# B&R Automation Studio project NewPendant_NG4_11_05_25A (part 9)

```c
			break;

			case 1: // Pulse

				curCfg->Param[parTIG_AmpSP].segmYes = 1;
				curCfg->Param[parTIG_AmpInSP].segmYes = 0;
				curCfg->Param[parTIG_AmpOutSP].segmYes = 0;
				curCfg->Param[parTIG_BackAmp].segmYes = 1;
				curCfg->Param[parTIG_PulseFreq].segmYes = 1;
				curCfg->Param[parTIG_PulseWidth].segmYes = 1;

				switch(curCfg->Param_ENUM[parENUM_AVC_Mode].val[0]){

					default:

					curCfg->Param[parAVC_VoltSP].segmYes = 1;
					curCfg->Param[parAVC_VoltInSP].segmYes = 0;
					curCfg->Param[parAVC_VoltOutSP].segmYes = 0;
					curCfg->Param[parAVC_VoltBackSP].segmYes = 1;

					break;

					case 1: // BackGround Locked

					curCfg->Param[parAVC_VoltSP].segmYes = 1;
					curCfg->Param[parAVC_VoltInSP].segmYes = 0;
					curCfg->Param[parAVC_VoltOutSP].segmYes = 0;
					curCfg->Param[parAVC_VoltBackSP].segmYes = 0;

					break;

					case 2: // ForeGround Locked

					curCfg->Param[parAVC_VoltSP].segmYes = 0;
					curCfg->Param[parAVC_VoltInSP].segmYes = 0;
					curCfg->Param[parAVC_VoltOutSP].segmYes = 0;
					curCfg->Param[parAVC_VoltBackSP].segmYes = 1;

					break;

					case 3: // Locked

					curCfg->Param[parAVC_VoltSP].segmYes = 0;
					curCfg->Param[parAVC_VoltInSP].segmYes = 0;
					curCfg->Param[parAVC_VoltOutSP].segmYes = 0;
					curCfg->Param[parAVC_VoltBackSP].segmYes = 0;

					break;

				}

			break;

			case 2: // Synch

				curCfg->Param[parTIG_AmpSP].segmYes = 1;
				curCfg->Param[parTIG_AmpInSP].segmYes = 0;
				curCfg->Param[parTIG_AmpOutSP].segmYes = 0;
				curCfg->Param[parTIG_BackAmp].segmYes = 1;
				curCfg->Param[parTIG_PulseFreq].segmYes = 0;
				curCfg->Param[parTIG_PulseWidth].segmYes = 0;

				switch(curCfg->Param_ENUM[parENUM_AVC_Mode].val[0]){

					default:

					curCfg->Param[parAVC_VoltSP].segmYes = 1;
					curCfg->Param[parAVC_VoltInSP].segmYes = 0;
					curCfg->Param[parAVC_VoltOutSP].segmYes = 0;
					curCfg->Param[parAVC_VoltBackSP].segmYes = 1;

					break;

					case 1: // BackGround Locked

					curCfg->Param[parAVC_VoltSP].segmYes = 1;
					curCfg->Param[parAVC_VoltInSP].segmYes = 0;
					curCfg->Param[parAVC_VoltOutSP].segmYes = 0;
					curCfg->Param[parAVC_VoltBackSP].segmYes = 0;

					break;

					case 2: // ForeGround Locked

					curCfg->Param[parAVC_VoltSP].segmYes = 0;
					curCfg->Param[parAVC_VoltInSP].segmYes = 0;
					curCfg->Param[parAVC_VoltOutSP].segmYes = 0;
					curCfg->Param[parAVC_VoltBackSP].segmYes = 1;

					break;

					case 3: // Locked

					curCfg->Param[parAVC_VoltSP].segmYes = 0;
					curCfg->Param[parAVC_VoltInSP].segmYes = 0;
					curCfg->Param[parAVC_VoltOutSP].segmYes = 0;
					curCfg->Param[parAVC_VoltBackSP].segmYes = 0;

					break;

				}

			break;

			case 3: // Synch In/Out

				curCfg->Param[parTIG_AmpSP].segmYes = 0;
				curCfg->Param[parTIG_AmpInSP].segmYes = 1;
				curCfg->Param[parTIG_AmpOutSP].segmYes = 1;
				curCfg->Param[parTIG_BackAmp].segmYes = 1;
				curCfg->Param[parTIG_PulseFreq].segmYes = 0;
				curCfg->Param[parTIG_PulseWidth].segmYes = 0;

				switch(curCfg->Param_ENUM[parENUM_AVC_Mode].val[0]){

					default:

					curCfg->Param[parAVC_VoltSP].segmYes = 0;
					curCfg->Param[parAVC_VoltInSP].segmYes = 1;
					curCfg->Param[parAVC_VoltOutSP].segmYes = 1;
					curCfg->Param[parAVC_VoltBackSP].segmYes = 1;

					break;

					case 1: // BackGround Locked

					curCfg->Param[parAVC_VoltSP].segmYes = 0;
					curCfg->Param[parAVC_VoltInSP].segmYes = 1;
					curCfg->Param[parAVC_VoltOutSP].segmYes = 1;
					curCfg->Param[parAVC_VoltBackSP].segmYes = 0;

					break;

					case 2: // ForeGround Locked

					curCfg->Param[parAVC_VoltSP].segmYes = 0;
					curCfg->Param[parAVC_VoltInSP].segmYes = 0;
					curCfg->Param[parAVC_VoltOutSP].segmYes = 0;
					curCfg->Param[parAVC_VoltBackSP].segmYes = 1;

					break;

					case 3: // Locked

					curCfg->Param[parAVC_VoltSP].segmYes = 0;
					curCfg->Param[parAVC_VoltInSP].segmYes = 0;
					curCfg->Param[parAVC_VoltOutSP].segmYes = 0;
					curCfg->Param[parAVC_VoltBackSP].segmYes = 0;

					break;

					}

			break;

		}

		switch(_TVL_MODE){

			default: // Straight

				curCfg->Param[parTVL_VelSP].segmYes = 1;
				curCfg->Param[parTVL_VelInSP].segmYes = 0;
				curCfg->Param[parTVL_VelOutSP].segmYes = 0;
				curCfg->Param[parTVL_VelBackSP].segmYes = 0;

			break;

			case 1:

				curCfg->Param[parTVL_VelSP].segmYes = 1;
				curCfg->Param[parTVL_VelInSP].segmYes = 0;
				curCfg->Param[parTVL_VelOutSP].segmYes = 0;
				curCfg->Param[parTVL_VelBackSP].segmYes = 1;

			break;

			case 2:

				curCfg->Param[parTVL_VelSP].segmYes = 0;
				curCfg->Param[parTVL_VelInSP].segmYes = 1;
				curCfg->Param[parTVL_VelOutSP].segmYes = 1;
				curCfg->Param[parTVL_VelBackSP].segmYes = 1;

			break;

		}

		switch(_WF_MODE){

			default: // Straight

				curCfg->Param[parWF_SpeedSP].segmYes = 1;
				curCfg->Param[parWF_SpeedInSP].segmYes = 0;
				curCfg->Param[parWF_SpeedOutSP].segmYes = 0;
				curCfg->Param[parWF_BkgSpeedSP].segmYes = 0;

			break;

			case 1:

				curCfg->Param[parWF_SpeedSP].segmYes = 1;
				curCfg->Param[parWF_SpeedInSP].segmYes = 0;
				curCfg->Param[parWF_SpeedOutSP].segmYes = 0;
				curCfg->Param[parWF_BkgSpeedSP].segmYes = 1;

			break;

			break;

			case 2:

				curCfg->Param[parWF_SpeedSP].segmYes = 0;
				curCfg->Param[parWF_SpeedInSP].segmYes = 1;
				curCfg->Param[parWF_SpeedOutSP].segmYes = 1;
				curCfg->Param[parWF_BkgSpeedSP].segmYes = 1;

			break;

			break;

		}

		switch(_WP_MODE){

			default: // Straight

				curCfg->Param[parWP_SpeedSP].segmYes = 1;
				curCfg->Param[parWP_SpeedInSP].segmYes = 0;
				curCfg->Param[parWP_SpeedOutSP].segmYes = 0;
				curCfg->Param[parWP_BkgSpeedSP].segmYes = 0;

			break;

			case 1:

				curCfg->Param[parWP_SpeedSP].segmYes = 1;
				curCfg->Param[parWP_SpeedInSP].segmYes = 0;
				curCfg->Param[parWP_SpeedOutSP].segmYes = 0;
				curCfg->Param[parWP_BkgSpeedSP].segmYes = 1;

			break;

			break;

			case 2:

				curCfg->Param[parWP_SpeedSP].segmYes = 0;
				curCfg->Param[parWP_SpeedInSP].segmYes = 1;
				curCfg->Param[parWP_SpeedOutSP].segmYes = 1;
				curCfg->Param[parWP_BkgSpeedSP].segmYes = 1;

			break;

			break;

		}

		hmi->PLC_Changes |= 0xF;
		KK_Was_Cahnged = 1;
	}

	_TIG_Mode = curCfg->Param_ENUM[parENUM_TIG_Mode].val[0];

	_AVC_Mode = curCfg->Param_ENUM[parENUM_AVC_Mode].val[0];

	_TVL_SYN_MODE = curCfg->Param_ENUM[parENUM_TVL_SYN_MODE].val[0];

	_WF_SYN_MODE = curCfg->Param_ENUM[parENUM_WF_SYN_MODE].val[0];

	_WP_SYN_MODE = curCfg->Param_ENUM[parENUM_WP_SYN_MODE].val[0];

	return;

}

void BumpParam(UINT param , SINT incr ){

	if(incr > 0)
		IncrParam(curCfg, param, m->curSegm[ZONE], 1.0);
	else
		DecrParam(curCfg, param, m->curSegm[ZONE], 1.0);

	if (! (curCalib->GenSetup[SETUP_WHERE_FILL] == 2)) //Not only Editor
		Fill_Segments(curCfg, param, m->curSegm[ZONE], curCalib->GenSetup[SETUP_AUTO_FILL],m->sm.Step);

	return;

}

void ChangeParam(UINT param , SINT incr ){

	switch(param){

		////////////////////////////////////////////
		case parTIG_AmpSP:

			switch(curCfg->Param_ENUM[parENUM_TIG_Mode].val[0]){

				default: // Straight

					BumpParam(parTIG_AmpSP , incr) ;

				break;

				case 1: // Pulse
				case 2: // Synch

					BumpParam(parTIG_AmpSP , incr) ;
					BumpParam(parTIG_BackAmp , incr) ;

				break;

				case 3: //Synch In/Out

					BumpParam(parTIG_AmpInSP , incr) ;
					BumpParam(parTIG_AmpOutSP , incr) ;
					BumpParam(parTIG_BackAmp , incr) ;

				break;

			}

		break;
		///////////////////////////////////////

		////////////////////////////////////////////
		case parTVL_VelSP:

			switch(curCfg->Param_ENUM[parENUM_TVL_SYN_MODE].val[0]){

				default: // Straight

					BumpParam(parTVL_VelSP , incr) ;

				break;

				case 1: // Synch

					if(curCfg->Param[parTVL_VelSP].val[m->curSegm[ZONE]] != 0.0)
						BumpParam(parTVL_VelSP , incr) ;

					if(curCfg->Param[parTVL_VelBackSP].val[m->curSegm[ZONE]] != 0.0)
						BumpParam(parTVL_VelBackSP , incr) ;

				break;

				case 2: //Synch In/Out

					if(curCfg->Param[parTVL_VelInSP].val[m->curSegm[ZONE]] != 0.0)
						BumpParam(parTVL_VelInSP , incr) ;

					if(curCfg->Param[parTVL_VelOutSP].val[m->curSegm[ZONE]] != 0.0)
						BumpParam(parTVL_VelOutSP , incr) ;

					if(curCfg->Param[parTVL_VelBackSP].val[m->curSegm[ZONE]] != 0.0)
						BumpParam(parTVL_VelBackSP , incr) ;

				break;

			}

		break;
		///////////////////////////////////////

		////////////////////////////////////////////
		case parWF_SpeedSP:

			switch(curCfg->Param_ENUM[parENUM_WF_SYN_MODE].val[0]){

				default: // Straight

					BumpParam(parWF_SpeedSP , incr) ;

				break;

				case 1: // Synch

					BumpParam(parWF_SpeedSP , incr) ;
					BumpParam(parWF_BkgSpeedSP , incr) ;

				break;

				case 2: //Synch In/Out

					BumpParam(parWF_SpeedInSP , incr) ;
					BumpParam(parWF_SpeedOutSP , incr) ;
					BumpParam(parWF_BkgSpeedSP , incr) ;

				break;

			}

		break;
		///////////////////////////////////////

		////////////////////////////////////////////
		case parWP_SpeedSP:

			switch(curCfg->Param_ENUM[parENUM_WP_SYN_MODE].val[0]){

				default: // Straight

					BumpParam(parWP_SpeedSP , incr) ;

				break;

				case 1: // Synch

					BumpParam(parWP_SpeedSP , incr) ;
					BumpParam(parWP_BkgSpeedSP , incr) ;

				break;

				case 2: //Synch In/Out

					BumpParam(parWP_SpeedInSP , incr) ;
					BumpParam(parWP_SpeedOutSP , incr) ;
					BumpParam(parWP_BkgSpeedSP , incr) ;

				break;

			}

		break;
		///////////////////////////////////////

		////////////////////////////////////////////
		case parAVC_VoltSP:

			switch(curCfg->Param_ENUM[parENUM_AVC_Mode].val[0]){

				case 0: // Continue

					switch(curCfg->Param_ENUM[parENUM_TIG_Mode].val[0]){

						default:

							BumpParam(parAVC_VoltSP , incr) ;

						break;

						case 1: //Pulse
						case 2: // Synch

							BumpParam(parAVC_VoltSP , incr) ;
							BumpParam(parAVC_VoltBackSP , incr) ;

						break;

						case 3: // Synch In/Out

							BumpParam(parAVC_VoltInSP , incr) ;
							BumpParam(parAVC_VoltOutSP , incr) ;
							BumpParam(parAVC_VoltBackSP , incr) ;

						break;

					}

				break;

				case 1: // Background Locked

					switch(curCfg->Param_ENUM[parENUM_TIG_Mode].val[0]){

						default:

							BumpParam(parAVC_VoltSP , incr) ;

						break;

						case 1: //Pulse
						case 2: // Synch

							BumpParam(parAVC_VoltSP , incr) ;

						break;

						case 3: // Synch In/Out

							BumpParam(parAVC_VoltInSP , incr) ;
							BumpParam(parAVC_VoltOutSP , incr) ;

						break;

					}

				break;

				case 2: // ForeGround Locked

					switch(curCfg->Param_ENUM[parENUM_TIG_Mode].val[0]){

						default:

							BumpParam(parAVC_VoltSP , incr) ;

						break;

						case 1: //Pulse
						case 2: // Synch
						case 3: // Synch In/Out

							BumpParam(parAVC_VoltBackSP , incr) ;

						break;

					}

				break;

			}

		break;
		///////////////////////////////////////

	}

	return;
}

void CalculateRunOverlap(){

	switch (curCfg->Param_ENUM[parENUM_TVL_MODE].val[0])
	{

		default: // relative

			Process[m->pCfg->HeadCfg.TVL.PROC_Indx].Param[0] = ((DINT) (curCfg->Param[parTVL_RunDist].val[0]) *m->ticksPerSegm); //Distance to	Run

			if(curCalib->GenSetup[SETUP_TWO_UP]> 0)
				Process[m->pCfg->HeadCfg.TVL.PROC_Indx].Param[3] = ((DINT) (curCfg->Param[parTVL_OverlapDist].val[0]) *m->ticksPerSegm); //Distance to	Rewrap
			else
				Process[m->pCfg->HeadCfg.TVL.PROC_Indx].Param[3] = ((DINT) (curCfg->Param[parTVL_RunDist].val[0] + curCfg->Param[parTVL_OverlapDist].val[0]) *m->ticksPerSegm); //Distance to  Rewrap

		break;

		case 1: // Side A overlap

			if (!m->ToolHeadID){

				Process[m->pCfg->HeadCfg.TVL.PROC_Indx].Param[0] = ((DINT) (curCfg->Param[parTVL_RunDist].val[0]) *m->ticksPerSegm); //Position to	Run

				if(curCalib->GenSetup[SETUP_TWO_UP]> 0)
					Process[m->pCfg->HeadCfg.TVL.PROC_Indx].Param[3] = ((DINT) (curCfg->Param[parTVL_OverlapDist].val[0]) *m->ticksPerSegm); //Position to	Rewrap
				else
					Process[m->pCfg->HeadCfg.TVL.PROC_Indx].Param[3] = ((DINT) (curCfg->Param[parTVL_RunDist].val[0] + curCfg->Param[parTVL_OverlapDist].val[0]) *m->ticksPerSegm); //Distance to  Rewrap

			}
			else{

				Process[m->pCfg->HeadCfg.TVL.PROC_Indx].Param[3] = 0;

				if(curCalib->GenSetup[SETUP_TWO_UP]> 0)
					Process[m->pCfg->HeadCfg.TVL.PROC_Indx].Param[0] = ((DINT) (curCfg->Param[parTVL_RunDist].val[0] - curCfg->Param[parTVL_OverlapDist].val[0]) *m->ticksPerSegm); //Position to	Run

				else
					Process[m->pCfg->HeadCfg.TVL.PROC_Indx].Param[0] = ((DINT) (curCfg->Param[parTVL_OverlapDist].val[0]) *m->ticksPerSegm)* (-1); //Position to	Run

			}

		break;

		case 2: // Side B overlap

			if (!m->ToolHeadID){

				Process[m->pCfg->HeadCfg.TVL.PROC_Indx].Param[0] = ((DINT) (curCfg->Param[parTVL_RunDist].val[0]- curCfg->Param[parTVL_OverlapDist].val[0]) *m->ticksPerSegm); //Distance to	Run

				if(curCalib->GenSetup[SETUP_TWO_UP]> 0)
					Process[m->pCfg->HeadCfg.TVL.PROC_Indx].Param[3] = 0; //Position to	Rewrap
				else
					Process[m->pCfg->HeadCfg.TVL.PROC_Indx].Param[3] = ((DINT) (curCfg->Param[parTVL_RunDist].val[0]) *m->ticksPerSegm); //Distance to  Rewrap

			}
			else{

				Process[m->pCfg->HeadCfg.TVL.PROC_Indx].Param[3] = ((DINT) (curCfg->Param[parTVL_OverlapDist].val[0]) *m->ticksPerSegm) ; //Distance to Run;

				if(curCalib->GenSetup[SETUP_TWO_UP]> 0)
					Process[m->pCfg->HeadCfg.TVL.PROC_Indx].Param[0] = ((DINT) (curCfg->Param[parTVL_RunDist].val[0]) *m->ticksPerSegm); //Distance to	Run

				else
					Process[m->pCfg->HeadCfg.TVL.PROC_Indx].Param[0] = 0; //Position to	Run

			}

		break;
	}

	/////////////////////////////////////////
	KK_ZigZag_Dist = curCfg->Param[parTVL_ZigZagDist].val[0];
	KK_Balance_Dist = curCfg->Param[parTVL_BalanceDist].val[0];

	if(KK_ZigZag_Dist != 0.0){

		if(curCalib->GenSetup[SETUP_ZIG_ZAG] == 0){

			if (!m->ToolHeadID){ // Head A

			}else{

				Process[m->pCfg->HeadCfg.TVL.PROC_Indx].Param[3] += (DINT)(KK_ZigZag_Dist *m->ticksPerSegm) ;

				curCalib->GenSetup[SETUP_ZIG_ZAG] = 1;

			}

		}else{

			if (!m->ToolHeadID){ // Head A

				Process[m->pCfg->HeadCfg.TVL.PROC_Indx].Param[0] += (DINT)(KK_ZigZag_Dist *m->ticksPerSegm);
				Process[m->pCfg->HeadCfg.TVL.PROC_Indx].Param[3] += (DINT)(KK_ZigZag_Dist *m->ticksPerSegm) ;

			}else{

				Process[m->pCfg->HeadCfg.TVL.PROC_Indx].Param[0] += (DINT)(KK_ZigZag_Dist *m->ticksPerSegm) ;

				curCalib->GenSetup[SETUP_ZIG_ZAG] = 0;

			}
		}

	}
	else
		curCalib->GenSetup[SETUP_ZIG_ZAG] = 0;

	///////////////////////////////////////////////////

	if (m->ToolHeadID)
		Process[m->pCfg->HeadCfg.TVL.PROC_Indx].Param[0] += (DINT)(KK_Balance_Dist *m->ticksPerSegm);

}

void SetTVL_Pos_Feedback(){

	if(curCalib->GenSetup[SETUP_TVL_SEC_ENC]){

		VectorStateMach[m->pCfg->HeadCfg.TVL.VECT_Indx].fParam[6] = 1.0;
		VectorStateMach[m->pCfg->HeadCfg.TVL.VECT_Indx].xCMD = VECT_Set_Param_6;

		TVL_ROT_Param_Set[0].EncPerTick = m->pCfg->HeadCfg.TVL.EncPerTick_SecEnc;

	}
	else{

		VectorStateMach[m->pCfg->HeadCfg.TVL.VECT_Indx].fParam[6] = 0.0;
		VectorStateMach[m->pCfg->HeadCfg.TVL.VECT_Indx].xCMD = VECT_Set_Param_6;

		TVL_ROT_Param_Set[0].EncPerTick = m->pCfg->HeadCfg.TVL.EncPerTick;
	}

return;

}

DINT Check_OSC_Amplt_and_Center(){
float pos;

	if(!OSC_TML_Param_Set[0].pVect || !OSC_TML_Param_Set[0].pPrimAmpl )
		return 0;

	if(OSC_TML_Param_Set[0].PosFbkIndx == 2)
		pos = OSC_TML_Param_Set[0].pVect->FbkVect.x2 ;

	else
		pos = OSC_TML_Param_Set[0].pVect->FbkVect.x ;

	if(((pos  + (*OSC_TML_Param_Set[0].pPrimAmpl)/2.0) > (OSC_TML_Param_Set[0].pVect->OutVect.softLimits[1] + 0.5))
		|| ((pos  - (*OSC_TML_Param_Set[0].pPrimAmpl)/2.0) < (OSC_TML_Param_Set[0].pVect->OutVect.softLimits[0] - 0.5))){

		strcpy(hmi->pMessage[0], "OSC Limits problem ");
		strcpy(hmi->pMessage[1], " ");
		xsprintf(hmi->pMessage[2], "Correct Amplitude");
		strcpy(hmi->pMessage[3], " or Position ?");

		//TimerStart(&hmi->MsgTmr, 1.0);

		hmi->xCMD = SHOW_POPUP_CMD;
		POPUP_EVENT = EVNT_OSC_ALLIGMENT;

		return 0;

	}
	return 1;
}

void CalculateRunOverlap_Cont(){

DINT mode;

	if((curCfg->Param_ENUM[parENUM_TVL_MODE].val[0] == 0 )
		|| (curCfg->Param_ENUM[parENUM_TVL_MODE].val[0] == 0 ))
		mode = 1; // Side A overlap
	else
		mode = curCfg->Param_ENUM[parENUM_TVL_MODE].val[0];

	switch (mode)
	{

		default: // relative

			Process[m->pCfg->HeadCfg.TVL.PROC_Indx].Param[0] = ((DINT) (curCfg->Param[parTVL_RunDist].val[0]) *m->ticksPerSegm); //Distance to	Run

			if((curCalib->GenSetup[SETUP_TWO_UP]> 0)&& 0)
				Process[m->pCfg->HeadCfg.TVL.PROC_Indx].Param[3] = ((DINT) (curCfg->Param[parTVL_OverlapDist].val[0]) *m->ticksPerSegm); //Distance to	Rewrap
			else
				Process[m->pCfg->HeadCfg.TVL.PROC_Indx].Param[3] = ((DINT) (curCfg->Param[parTVL_RunDist].val[0] + curCfg->Param[parTVL_OverlapDist].val[0]) *m->ticksPerSegm); //Distance to  Rewrap

		break;

		case 1: // Side A overlap

			if (!m->ToolHeadID){

				Process[m->pCfg->HeadCfg.TVL.PROC_Indx].Param[0] = ((DINT) (curCfg->Param[parTVL_RunDist].val[0]) *m->ticksPerSegm); //Position to	Run

				if((curCalib->GenSetup[SETUP_TWO_UP]> 0)&& 0)
					Process[m->pCfg->HeadCfg.TVL.PROC_Indx].Param[3] = ((DINT) (curCfg->Param[parTVL_OverlapDist].val[0]) *m->ticksPerSegm); //Position to	Rewrap
				else
					Process[m->pCfg->HeadCfg.TVL.PROC_Indx].Param[3] = ((DINT) (curCfg->Param[parTVL_RunDist].val[0] + curCfg->Param[parTVL_OverlapDist].val[0]) *m->ticksPerSegm); //Distance to  Rewrap

			}
			else{

				Process[m->pCfg->HeadCfg.TVL.PROC_Indx].Param[3] = 0;

				if((curCalib->GenSetup[SETUP_TWO_UP]> 0)&& 0)
					Process[m->pCfg->HeadCfg.TVL.PROC_Indx].Param[0] = ((DINT) (curCfg->Param[parTVL_RunDist].val[0] - curCfg->Param[parTVL_OverlapDist].val[0]) *m->ticksPerSegm); //Position to	Run

				else
					Process[m->pCfg->HeadCfg.TVL.PROC_Indx].Param[0] = ((DINT) (curCfg->Param[parTVL_OverlapDist].val[0]) *m->ticksPerSegm)* (-1); //Position to	Run

			}

		break;

		case 2: // Side B overlap

			if (!m->ToolHeadID){

				Process[m->pCfg->HeadCfg.TVL.PROC_Indx].Param[0] = ((DINT) (curCfg->Param[parTVL_RunDist].val[0]- curCfg->Param[parTVL_OverlapDist].val[0]) *m->ticksPerSegm); //Distance to	Run

				if((curCalib->GenSetup[SETUP_TWO_UP]> 0)&& 0)
					Process[m->pCfg->HeadCfg.TVL.PROC_Indx].Param[3] = 0; //Position to	Rewrap
				else
					Process[m->pCfg->HeadCfg.TVL.PROC_Indx].Param[3] = ((DINT) (curCfg->Param[parTVL_RunDist].val[0]) *m->ticksPerSegm); //Distance to  Rewrap

			}
			else{

				Process[m->pCfg->HeadCfg.TVL.PROC_Indx].Param[3] = ((DINT) (curCfg->Param[parTVL_OverlapDist].val[0]) *m->ticksPerSegm) ; //Distance to Run;

				if((curCalib->GenSetup[SETUP_TWO_UP]> 0)&& 0)
					Process[m->pCfg->HeadCfg.TVL.PROC_Indx].Param[0] = ((DINT) (curCfg->Param[parTVL_RunDist].val[0]) *m->ticksPerSegm); //Distance to	Run

				else
					Process[m->pCfg->HeadCfg.TVL.PROC_Indx].Param[0] = 0; //Position to	Run

			}

		break;
	}

}

void CalculateRunOverlap_Cont_OneWay(){

DINT mode;

	if((curCfg->Param_ENUM[parENUM_TVL_MODE].val[0] == 0 )
		|| (curCfg->Param_ENUM[parENUM_TVL_MODE].val[0] == 0 ))
		mode = 1; // Side A overlap
	else
		mode = curCfg->Param_ENUM[parENUM_TVL_MODE].val[0];

	switch (mode)
	{

		default: // relative

			Process[m->pCfg->HeadCfg.TVL.PROC_Indx].Param[0] = ((DINT) (curCfg->Param[parTVL_RunDist].val[0]) *m->ticksPerSegm); //Distance to	Run

			if((curCalib->GenSetup[SETUP_TWO_UP]> 0) || 1)
				Process[m->pCfg->HeadCfg.TVL.PROC_Indx].Param[3] = ((DINT) (curCfg->Param[parTVL_OverlapDist].val[0]) *m->ticksPerSegm); //Distance to	Rewrap
			else
				Process[m->pCfg->HeadCfg.TVL.PROC_Indx].Param[3] = ((DINT) (curCfg->Param[parTVL_RunDist].val[0] + curCfg->Param[parTVL_OverlapDist].val[0]) *m->ticksPerSegm); //Distance to  Rewrap

		break;

		case 1: // Side A overlap

			if (!m->ToolHeadID){

				Process[m->pCfg->HeadCfg.TVL.PROC_Indx].Param[0] = ((DINT) (curCfg->Param[parTVL_RunDist].val[0]) *m->ticksPerSegm); //Position to	Run

				if((curCalib->GenSetup[SETUP_TWO_UP]> 0) || 1)
					Process[m->pCfg->HeadCfg.TVL.PROC_Indx].Param[3] = ((DINT) (curCfg->Param[parTVL_OverlapDist].val[0]) *m->ticksPerSegm); //Position to	Rewrap
				else
					Process[m->pCfg->HeadCfg.TVL.PROC_Indx].Param[3] = ((DINT) (curCfg->Param[parTVL_RunDist].val[0] + curCfg->Param[parTVL_OverlapDist].val[0]) *m->ticksPerSegm); //Distance to  Rewrap

			}
			else{

				Process[m->pCfg->HeadCfg.TVL.PROC_Indx].Param[3] = 0;

				if((curCalib->GenSetup[SETUP_TWO_UP]> 0) || 1)
					Process[m->pCfg->HeadCfg.TVL.PROC_Indx].Param[0] = ((DINT) (curCfg->Param[parTVL_RunDist].val[0] - curCfg->Param[parTVL_OverlapDist].val[0]) *m->ticksPerSegm); //Position to	Run

				else
					Process[m->pCfg->HeadCfg.TVL.PROC_Indx].Param[0] = ((DINT) (curCfg->Param[parTVL_OverlapDist].val[0]) *m->ticksPerSegm)* (-1); //Position to	Run

			}

		break;

		case 2: // Side B overlap

			if (!m->ToolHeadID){

				Process[m->pCfg->HeadCfg.TVL.PROC_Indx].Param[0] = ((DINT) (curCfg->Param[parTVL_RunDist].val[0]- curCfg->Param[parTVL_OverlapDist].val[0]) *m->ticksPerSegm); //Distance to	Run

				if((curCalib->GenSetup[SETUP_TWO_UP]> 0) || 1)
					Process[m->pCfg->HeadCfg.TVL.PROC_Indx].Param[3] = 0; //Position to	Rewrap
				else
					Process[m->pCfg->HeadCfg.TVL.PROC_Indx].Param[3] = ((DINT) (curCfg->Param[parTVL_RunDist].val[0]) *m->ticksPerSegm); //Distance to  Rewrap

			}
			else{

				Process[m->pCfg->HeadCfg.TVL.PROC_Indx].Param[3] = ((DINT) (curCfg->Param[parTVL_OverlapDist].val[0]) *m->ticksPerSegm) ; //Distance to Run;

				if((curCalib->GenSetup[SETUP_TWO_UP]> 0) || 1)
					Process[m->pCfg->HeadCfg.TVL.PROC_Indx].Param[0] = ((DINT) (curCfg->Param[parTVL_RunDist].val[0]) *m->ticksPerSegm); //Distance to	Run

				else
					Process[m->pCfg->HeadCfg.TVL.PROC_Indx].Param[0] = 0; //Position to	Run

			}

		break;
	}

/*
	{

		default: // relative

			Process[m->pCfg->HeadCfg.TVL.PROC_Indx].Param[0] = ((DINT) (curCfg->Param[parTVL_RunDist].val[0]) *m->ticksPerSegm); //Distance to	Run

			if(curCalib->GenSetup[SETUP_TWO_UP]> 0)
				Process[m->pCfg->HeadCfg.TVL.PROC_Indx].Param[3] = ((DINT) (curCfg->Param[parTVL_OverlapDist].val[0]) *m->ticksPerSegm); //Distance to	Rewrap
			else
				Process[m->pCfg->HeadCfg.TVL.PROC_Indx].Param[3] = ((DINT) (curCfg->Param[parTVL_RunDist].val[0] + curCfg->Param[parTVL_OverlapDist].val[0]) *m->ticksPerSegm); //Distance to  Rewrap

		break;

		case 1: // Side A overlap

			if (!m->ToolHeadID){

				Process[m->pCfg->HeadCfg.TVL.PROC_Indx].Param[0] = ((DINT) (curCfg->Param[parTVL_RunDist].val[0]) *m->ticksPerSegm); //Position to	Run

				if(curCalib->GenSetup[SETUP_TWO_UP]> 0)
					Process[m->pCfg->HeadCfg.TVL.PROC_Indx].Param[3] = ((DINT) (curCfg->Param[parTVL_OverlapDist].val[0]) *m->ticksPerSegm); //Position to	Rewrap
				else
					Process[m->pCfg->HeadCfg.TVL.PROC_Indx].Param[3] = ((DINT) (curCfg->Param[parTVL_RunDist].val[0] + curCfg->Param[parTVL_OverlapDist].val[0]) *m->ticksPerSegm); //Distance to  Rewrap

			}
			else{

				Process[m->pCfg->HeadCfg.TVL.PROC_Indx].Param[3] = 0;

				if(curCalib->GenSetup[SETUP_TWO_UP]> 0)
					Process[m->pCfg->HeadCfg.TVL.PROC_Indx].Param[0] = ((DINT) (curCfg->Param[parTVL_RunDist].val[0] - curCfg->Param[parTVL_OverlapDist].val[0]) *m->ticksPerSegm); //Position to	Run

				else
					Process[m->pCfg->HeadCfg.TVL.PROC_Indx].Param[0] = ((DINT) (curCfg->Param[parTVL_OverlapDist].val[0]) *m->ticksPerSegm)* (-1); //Position to	Run

			}

		break;

		case 2: // Side B overlap

			if (!m->ToolHeadID){

				Process[m->pCfg->HeadCfg.TVL.PROC_Indx].Param[0] = ((DINT) (curCfg->Param[parTVL_RunDist].val[0]- curCfg->Param[parTVL_OverlapDist].val[0]) *m->ticksPerSegm); //Distance to	Run

				if(curCalib->GenSetup[SETUP_TWO_UP]> 0)
					Process[m->pCfg->HeadCfg.TVL.PROC_Indx].Param[3] = 0; //Position to	Rewrap
				else
					Process[m->pCfg->HeadCfg.TVL.PROC_Indx].Param[3] = ((DINT) (curCfg->Param[parTVL_RunDist].val[0]) *m->ticksPerSegm); //Distance to  Rewrap

			}
			else{

				Process[m->pCfg->HeadCfg.TVL.PROC_Indx].Param[3] = ((DINT) (curCfg->Param[parTVL_OverlapDist].val[0]) *m->ticksPerSegm) ; //Distance to Run;

				if(curCalib->GenSetup[SETUP_TWO_UP]> 0)
					Process[m->pCfg->HeadCfg.TVL.PROC_Indx].Param[0] = ((DINT) (curCfg->Param[parTVL_RunDist].val[0]) *m->ticksPerSegm); //Distance to	Run

				else
					Process[m->pCfg->HeadCfg.TVL.PROC_Indx].Param[0] = 0; //Position to	Run

			}

		break;
	}
*/
}

void RestartStateMach(){
int i;

#ifdef 	MIG_EXP_SYSTEM

	switch(TML_Restart_Step){

		case 0:

		break;

		case 1:

			TML_Restart_Indx = 0;

			Kick_TML_Cmd = 1;

			TML_MTR_INST[TML_AX_WRST].Disable = 1;
			VectorStateMach[VECT_WRST].simul = 1;
			VectorStateMach[VECT_WRST].testMode = 1;

			TimerStart(&Restart_Tmr, 0.5);

			TML_Restart_Step++;

		break;

		case 2:

			if(!TimerIsTimeOut(&Restart_Tmr))
				break;

			if(TML_Restart_Indx < TML_SERVO_NUM ){

				if(!TML_MTR_INST[TML_Restart_Indx].Disable && TML_MTR_INST[TML_Restart_Indx].pState
					&&(Kick_TML_Cmd == 0)){

					TML_MTR_INST[TML_Restart_Indx].xCMD = TML_RESTART;
					TML_Restart_Step++;

				}
				else
					TML_Restart_Indx++;

			}
			else
				TML_Restart_Step = 10;

		break;

		case 3:

			if((TML_MTR_INST[TML_Restart_Indx].xCMD == 0)
				|| (TML_MTR_INST[TML_Restart_Indx].xCMD == 255) // Error
				|| (TML_MTR_INST[TML_Restart_Indx].xCMD == TML_WAIT_FOR_DOWNLOAD)
				){

				TML_Restart_Indx++;
				//Kick_TML_Cmd = 1;

				TimerStart(&Restart_Tmr, 0.8);
				TML_Restart_Step = 2;
				//TML_Restart_Step = 4;
			}

		break;

		case 4:

		break;

		case 10:

			for (i = 0; i < PROCESS_NUM; i++){

				if(i == m->pCfg->HeadCfg.GAS.PROC_Indx)
					Process[i].xCMD = prcsSTOP;
				else
					Process[i].xCMD = prcsRESTART;

			}

			TML_Restart_Step = 0;

		break;

	}

	TimerExecute(&Restart_Tmr);
#else

/*

for (i = 0; i < PROCESS_NUM; i++)
	Process[i].xCMD = prcsRESTART;

for (i = 0; i < TML_SERVO_NUM; i++)
{

	TML_MTR_INST[i].xCMD = TML_RESTART;
	TML_MTR_INST[i]._int.restartCnt = 0;
	TML_MTR_INST[i]._int.Init = 0;
}
*/

	switch(TML_Restart_Step){

		case 0:

		break;

		case 1:

			TML_Restart_Indx = 0;

			TML_Restart_Step++;

		break;

		case 2:

			if(TML_Restart_Indx < TML_SERVO_NUM ){

				if(!TML_MTR_INST[TML_Restart_Indx].Disable && TML_MTR_INST[TML_Restart_Indx].pState){

					TML_MTR_INST[TML_Restart_Indx].xCMD = TML_RESTART;
					TML_Restart_Step++;

				}
				else
					TML_Restart_Indx++;

			}
			else
				TML_Restart_Step = 10;

		break;

		case 3:

			TML_Restart_Indx++;
			TML_Restart_Step = 2;

		break;

		case 10:

			for (i = 0; i < PROCESS_NUM; i++){

				if(i == m->pCfg->HeadCfg.GAS.PROC_Indx)
					Process[i].xCMD = prcsSTOP;
				else
					Process[i].xCMD = prcsRESTART;

			}

			TML_Restart_Step = 0;

		break;

	}

	switch(Process_Restart_Step){

	}

#endif

}

plcbit Find_ext_txt(char *name , char* ext){
UINT len , ext_len;

		len = strlen(name);

		ext_len = strlen(ext);

		if(len >= ext_len){

			if(strcmp(&name[len-ext_len] ,ext) == 0)
				return 1;
			else
				return 0;

		}
		else
			return 0;

}

void FourAxisTIG(){

int i;

	for (i = 0 ; i < 2 ; i++){

		/**   Instances and pointer population **/
		pMaster[i] = &Master[i];
		pLCD_MGR[i] = &LCD_MGR[i];
		pRS232[i] = &RS232[i];
		pPendant[i] = &Pendant[i];

		strcpy(Pendant[i].RSDeviceStr , "IF1");

		// To jest nadal w SuperMaster dla Androida
		/*
		pMaster[i]->pNode[i] = (UDINT)&NODES[i];
		pMaster[i]->pUnits = Units;
		*/

		pMaster[i]->pCfg = &Cfg;
		pMaster[i]->pCurCfg = &CurCfg;
		pMaster[i]->pCalib = &CurCalib;
		pMaster[i]->pDefaultCalib = &DefaultCalib;
		//pMaster[i]->pLog =&ErrorMgr;
		pMaster[i]->pScaledUnitIndx = curScaledUnitIndx;
		//pMaster[i]->pScaledVar = (UDINT)ScaledVar;
		pMaster[i]->pScaledVar = (UDINT)&Cfg.ScaledVar;
		pMaster[i]->pSegmentTable = (UDINT)&SegmentsTable;
		//pMaster[i]->pProc = Process;

		pMaster[i]->xCmd = mstrRESTART;
		pMaster[i]->Active = 0;

	}

	/***************************/
	//  Assigment to Hot Wire hardware must be here

	for (i = 0 ; i < 4 ; i++){

		DC_Mtr[i].Hrdw.pPulseWidthPWM = &motors[i].Hardware.PulseWidthPWM;
		DC_Mtr[i].Hrdw.pEncFbk = &motors[i].Hardware.Counter;
		//Hardware[i].PWM[0].PeriodDurationPWM = &motors[i].Hardware.PeriodDurationPWM ;

	}

	#ifdef SYSTEM_SIMULATION

		Master[0].pESTOP_Inp = 0;
		Master[0].ESTOP = 0;

		Master[1].pESTOP_Inp = 0;
		Master[1].ESTOP = 0;

	#else

		Master[0].pESTOP_Inp = &hardware.Inputs[5]; //ControlModule_Estop_Active
		Master[1].pESTOP_Inp = &hardware.Inputs[5]; //ControlModule_Estop_Active

	#endif

	// working with MPC only
	Master[0].pESTOP_Out = &hardware.Outputs[7]; //ControlModule_Estop_LOOP contact

	HW_PS_Param_Set[0].pAnal_Output 	= &hardware.AnalogOutputs[1]; // HotwirePS_AO
	HW_PS_Param_Set[0].pOutput			= &hardware.Outputs[2]; //HotwirePS_Enable

	PS_Param_Set[0].pAnal_Output 	= &hardware.AnalogOutputs[0];  //PrimaryPS_AO positive
	// Check in Head Configuration also
	PS_Param_Set[0].pAnal_Output_neg = &hardware.AnalogOutputs[3];  //PrimaryPS_AO negative

	PS_Param_Set[0].pOutput			= &hardware.Outputs[0]; //PrimaryPS_Enable

	/***************************/

return;
}
```
